TYPE st_Data :
STRUCT
	x	: INT;
	y	: INT;
END_STRUCT
END_TYPE

(* stored: Version 1.1.0.1
   DUT st_Data: Id {3550f400-31d2-4f6c-bd75-12d4af6897e6} *)
